// TIA Portal project "Proyecto_iolink" (V16)

(* hardware
DEVICE "S7-1200 station_1"  S7-1200 Station
   slot 0: "Rack_0"  S7-1200 Rack  Rack  V1.0
   slot 1: "PLC_1"  CPU 1215C DC/DC/DC  6ES7 215-1AG40-0XB0  V4.4
DEVICE "ET 200SP station_1"  ET 200SP-Station
   slot 0: "Rack_0"  Rack  6ES5 710-8MAx1
   slot 0: "IO-Device_1"  IM 155-6 PN/2 HF  6ES7 155-6AU01-0CN0  V4.2
   slot 1: "CM 4xIO-Link_1"  CM 4xIO-Link  6ES7 137-6BD00-0BA0  V2.2
      slot 1: "CM 4xIO-Link_1"  6ES7 137-6BD00-0BA0
   slot 2: "DI 8x24VDC HF_1"  DI 8x24VDC HF  6ES7 131-6BF00-0CA0  V2.0
      slot 1: "DI 8x24VDC HF_1"  DI 8x24VDC HF
   slot 3: "DI 8x24VDC HF_2"  DI 8x24VDC HF  6ES7 131-6BF00-0CA0  V2.0
      slot 1: "DI 8x24VDC HF_2"  DI 8x24VDC HF
   slot 4: "DQ 8x24VDC/0.5A HF_1"  DQ 8x24VDC/0.5A HF  6ES7 132-6BF00-0CA0  V2.0
      slot 1: "DQ 8x24VDC/0.5A HF_1"  DQ 8x24VDC/0.5A HF
   slot 5: "DQ 8x24VDC/0.5A HF_2"  DQ 8x24VDC/0.5A HF  6ES7 132-6BF00-0CA0  V2.0
      slot 1: "DQ 8x24VDC/0.5A HF_2"  DQ 8x24VDC/0.5A HF
   slot 6: "Módulo servidor_1"  Server module  6ES7 193-6PA00-0AA0  V1.1
      slot 1: "Módulo servidor_1"  Server module
   slot 127: "BA 2xRJ45"  BA 2xRJ45  6ES7 193-6AR00-0AA0  V0.0
      slot 1: "Port_1"  X1 P1 R  6ES7 193-6AR00-0AA0  V0.0
      slot 2: "Port_2"  X1 P2 R  6ES7 193-6AR00-0AA0  V0.0
*)

// ===== PLC "PLC_1"  CPU 1215C DC/DC/DC =====

VAR_GLOBAL   // PLC tag table "Tabla de variables estándar"
   "interruptor" AT %I34.0 : Bool;
   "piloto" AT %Q35.0 : Bool;
   "detectando_sensor_capacitivo" AT %I3.0 : Bool;
   "distancia_sensor_capacitivo" AT %IW2 : Int;
   "baliza" AT %Q2.0 : "PIQ - BNI IOL-800-000-Z036";
   "configuracion_baliza" AT %QB2 : Byte;
END_VAR

TYPE "PII - KI6000"
   STRUCT
      "Datos del proceso de entrada/salida - PDV1 (Invalid Data Type)" : Bool;
      "Reserved Bit" : Bool;
      "Reserved Bit_1" : Bool;
      "Reserved Bit_2" : Bool;
      "Reserved Bit_3" : Bool;
      "Reserved Bit_4" : Bool;
      "Reserved Bit_5" : Bool;
      "Reserved Bit_6" : Bool;
      "Datos del proceso de entrada/salida - BDC1" : Bool;
      "Reserved Bit_7" : Bool;
      "Reserved Bit_8" : Bool;
      "Reserved Bit_9" : Bool;
      "Reserved Bit_10" : Bool;
      "Reserved Bit_11" : Bool;
      "Reserved Bit_12" : Bool;
      "Reserved Bit_13" : Bool;
   END_STRUCT;
END_TYPE

TYPE "PIQ - BNI IOL-800-000-Z036"
   STRUCT
      "Process Data Out - Color of segment 1 (Invalid Data Type)" : Bool;
      "Reserved Bit" : Bool;
      "Reserved Bit_1" : Bool;
      "Process Data Out - Segment 1 blinks" : Bool;
      "Reserved Bit_2" : Bool;
      "Process Data Out - Sync Start" : Bool;
      "Process Data Out - Sync Impulse" : Bool;
   END_STRUCT;
END_TYPE

DATA_BLOCK "Variables"   // DB1
{ S7_Optimized_Access := 'TRUE' }
VERSION : 0.1
   VAR
      distancia_mm : Int;
   END_VAR
BEGIN
END_DATA_BLOCK

ORGANIZATION_BLOCK "Main"   // OB1, LAD, ProgramCycle
TITLE = "Main Program Sweep (Cycle)"
{ S7_Optimized_Access := 'TRUE' }
VERSION : 0.1
   VAR_INPUT
      Initial_Call : Bool;   // Initial call of this OB
      Remanence : Bool;   // =True, if remanent data are available
   END_VAR
BEGIN

REGION Network 1
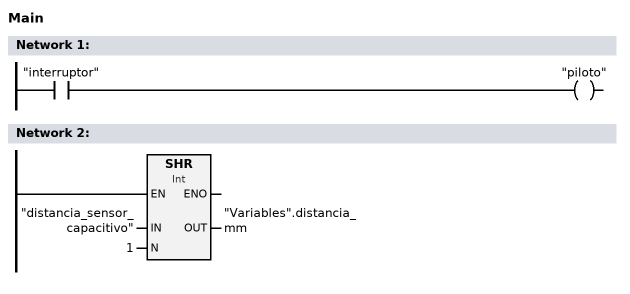
   RUNG wire#powerrail
      Contact( "interruptor" )
      Coil( "piloto" )
   END_RUNG
   // the same network as SCL:
   "piloto" := "interruptor";
END_REGION

REGION Network 2
   RUNG wire#powerrail
      { S7_Templates := "SrcType := Int" } Shr(in := "distancia_sensor_capacitivo", n := 1, out => "Variables".distancia_mm)
   END_RUNG
   // the same network as SCL:
   "Variables".distancia_mm := SHR(IN := "distancia_sensor_capacitivo", N := 1);
END_REGION
END_ORGANIZATION_BLOCK